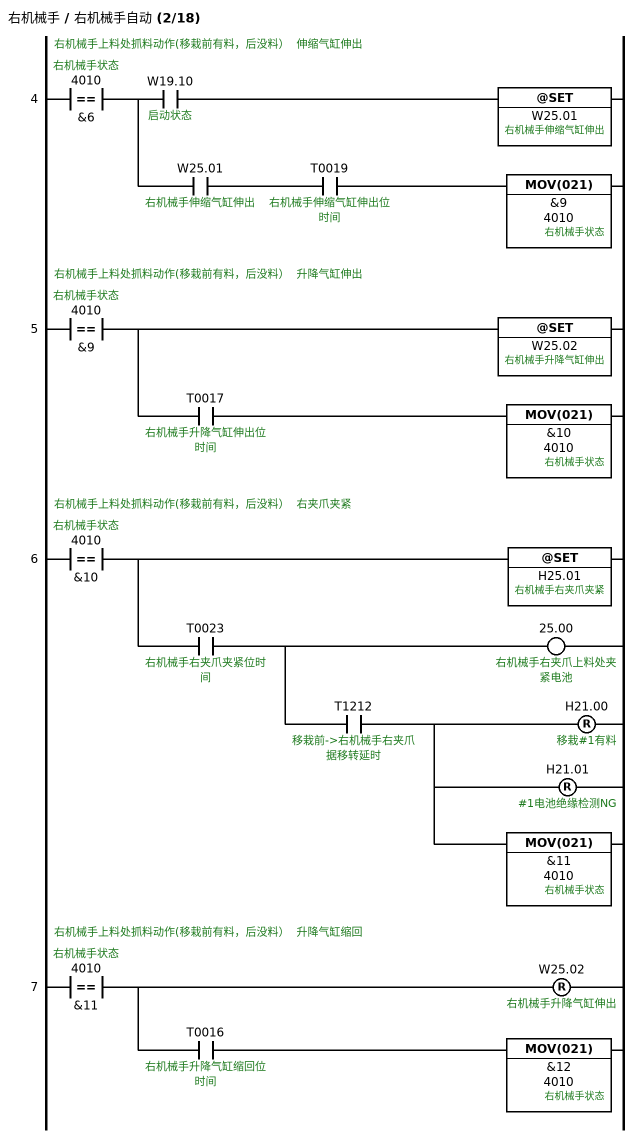
; rung 4: 右机械手上料处抓料动作(移栽前有料，后没料）  伸缩气缸伸出
LD=(300) 4010 &6  ; 右机械手状态
OUT TR0
AND W19.10  ; 启动状态
@SET W25.01  ; 右机械手伸缩气缸伸出
LD TR0
AND W25.01  ; 右机械手伸缩气缸伸出
AND T0019  ; 右机械手伸缩气缸伸出位时间
MOV(021) &9 4010  ; 右机械手状态
; rung 5: 右机械手上料处抓料动作(移栽前有料，后没料）  升降气缸伸出
LD=(300) 4010 &9  ; 右机械手状态
@SET W25.02  ; 右机械手升降气缸伸出
AND T0017  ; 右机械手升降气缸伸出位时间
MOV(021) &10 4010  ; 右机械手状态
; rung 6: 右机械手上料处抓料动作(移栽前有料，后没料）  右夹爪夹紧
LD=(300) 4010 &10  ; 右机械手状态
@SET H25.01  ; 右机械手右夹爪夹紧
AND T0023  ; 右机械手右夹爪夹紧位时间
OUT 25.00  ; 右机械手右夹爪上料处夹紧电池
AND T1212  ; 移栽前->右机械手右夹爪据移转延时
RSET H21.00  ; 移栽#1有料
RSET H21.01  ; #1电池绝缘检测NG
MOV(021) &11 4010  ; 右机械手状态
; rung 7: 右机械手上料处抓料动作(移栽前有料，后没料）  升降气缸缩回
LD=(300) 4010 &11  ; 右机械手状态
RSET W25.02  ; 右机械手升降气缸伸出
AND T0016  ; 右机械手升降气缸缩回位时间
MOV(021) &12 4010  ; 右机械手状态

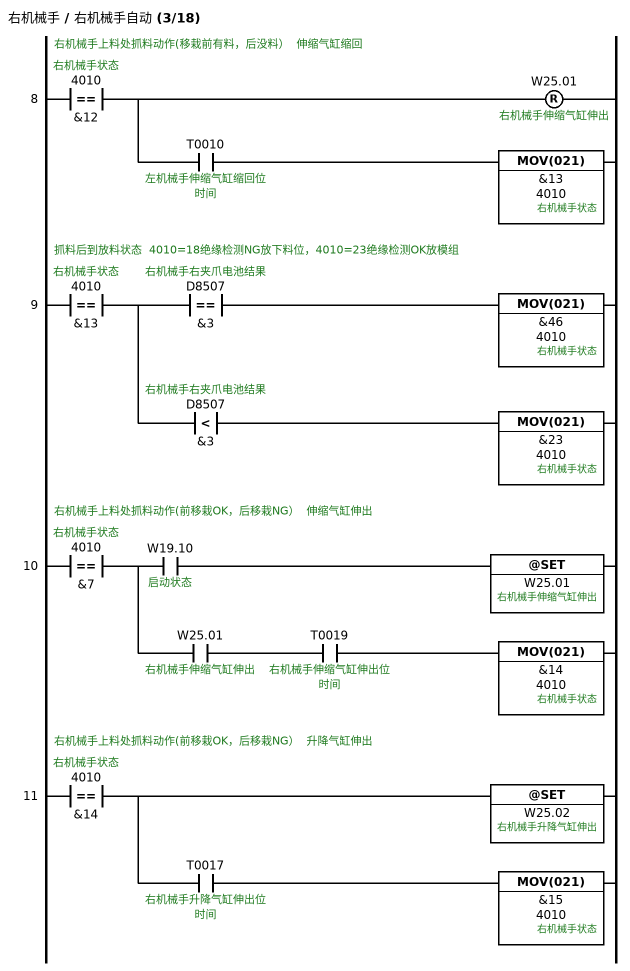
; rung 8: 右机械手上料处抓料动作(移栽前有料，后没料）  伸缩气缸缩回
LD=(300) 4010 &12  ; 右机械手状态
RSET W25.01  ; 右机械手伸缩气缸伸出
AND T0010  ; 左机械手伸缩气缸缩回位时间
MOV(021) &13 4010  ; 右机械手状态
; rung 9: 抓料后到放料状态  4010=18绝缘检测NG放下料位，4010=23绝缘检测OK放模组
LD=(300) 4010 &13  ; 右机械手状态
OUT TR0
AND=(300) D8507 &3  ; 右机械手右夹爪电池结果
MOV(021) &46 4010  ; 右机械手状态
LD TR0
AND<(310) D8507 &3  ; 右机械手右夹爪电池结果
MOV(021) &23 4010  ; 右机械手状态
; rung 10: 右机械手上料处抓料动作(前移栽OK，后移栽NG）  伸缩气缸伸出
LD=(300) 4010 &7  ; 右机械手状态
OUT TR0
AND W19.10  ; 启动状态
@SET W25.01  ; 右机械手伸缩气缸伸出
LD TR0
AND W25.01  ; 右机械手伸缩气缸伸出
AND T0019  ; 右机械手伸缩气缸伸出位时间
MOV(021) &14 4010  ; 右机械手状态
; rung 11: 右机械手上料处抓料动作(前移栽OK，后移栽NG）  升降气缸伸出
LD=(300) 4010 &14  ; 右机械手状态
@SET W25.02  ; 右机械手升降气缸伸出
AND T0017  ; 右机械手升降气缸伸出位时间
MOV(021) &15 4010  ; 右机械手状态

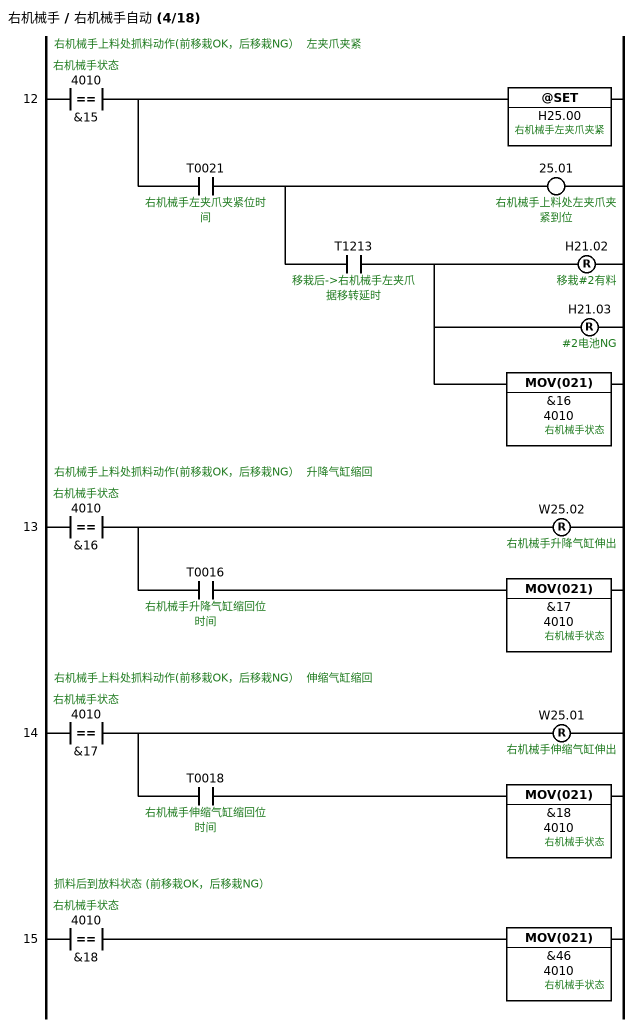
; rung 12: 右机械手上料处抓料动作(前移栽OK，后移栽NG）  左夹爪夹紧
LD=(300) 4010 &15  ; 右机械手状态
@SET H25.00  ; 右机械手左夹爪夹紧
AND T0021  ; 右机械手左夹爪夹紧位时间
OUT 25.01  ; 右机械手上料处左夹爪夹紧到位
AND T1213  ; 移栽后->右机械手左夹爪据移转延时
RSET H21.02  ; 移栽#2有料
RSET H21.03  ; #2电池NG
MOV(021) &16 4010  ; 右机械手状态
; rung 13: 右机械手上料处抓料动作(前移栽OK，后移栽NG）  升降气缸缩回
LD=(300) 4010 &16  ; 右机械手状态
RSET W25.02  ; 右机械手升降气缸伸出
AND T0016  ; 右机械手升降气缸缩回位时间
MOV(021) &17 4010  ; 右机械手状态
; rung 14: 右机械手上料处抓料动作(前移栽OK，后移栽NG）  伸缩气缸缩回
LD=(300) 4010 &17  ; 右机械手状态
RSET W25.01  ; 右机械手伸缩气缸伸出
AND T0018  ; 右机械手伸缩气缸缩回位时间
MOV(021) &18 4010  ; 右机械手状态
; rung 15: 抓料后到放料状态 (前移栽OK，后移栽NG）
LD=(300) 4010 &18  ; 右机械手状态
MOV(021) &46 4010  ; 右机械手状态

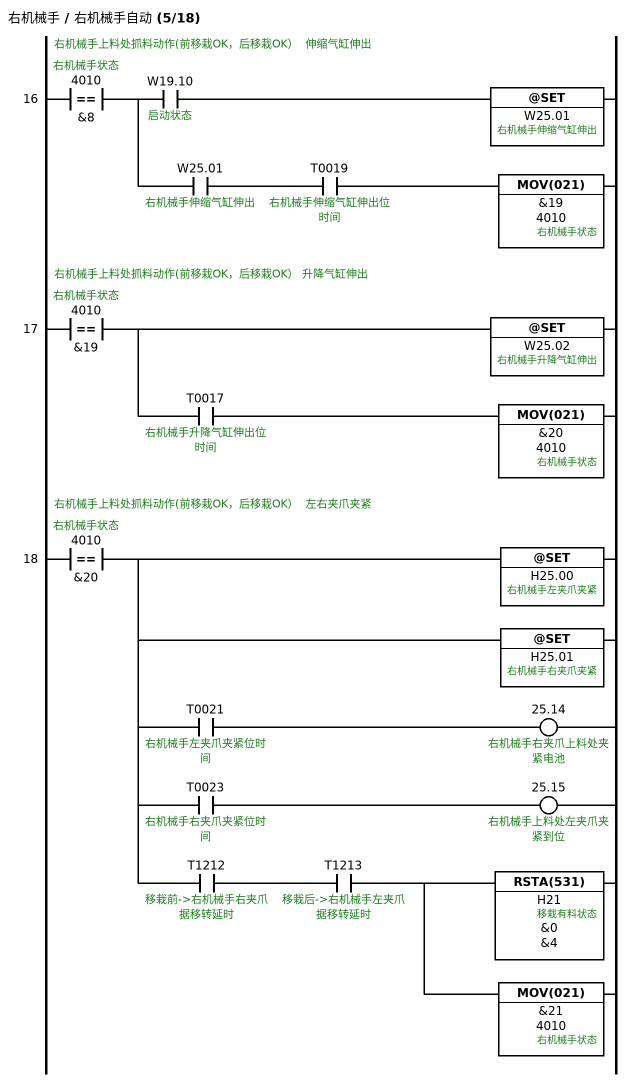
; rung 16: 右机械手上料处抓料动作(前移栽OK，后移栽OK）  伸缩气缸伸出
LD=(300) 4010 &8  ; 右机械手状态
OUT TR0
AND W19.10  ; 启动状态
@SET W25.01  ; 右机械手伸缩气缸伸出
LD TR0
AND W25.01  ; 右机械手伸缩气缸伸出
AND T0019  ; 右机械手伸缩气缸伸出位时间
MOV(021) &19 4010  ; 右机械手状态
; rung 17: 右机械手上料处抓料动作(前移栽OK，后移栽OK） 升降气缸伸出
LD=(300) 4010 &19  ; 右机械手状态
@SET W25.02  ; 右机械手升降气缸伸出
AND T0017  ; 右机械手升降气缸伸出位时间
MOV(021) &20 4010  ; 右机械手状态
; rung 18: 右机械手上料处抓料动作(前移栽OK，后移栽OK）  左右夹爪夹紧
LD=(300) 4010 &20  ; 右机械手状态
OUT TR0
@SET H25.00  ; 右机械手左夹爪夹紧
@SET H25.01  ; 右机械手右夹爪夹紧
AND T0021  ; 右机械手左夹爪夹紧位时间
OUT 25.14  ; 右机械手右夹爪上料处夹紧电池
LD TR0
AND T0023  ; 右机械手右夹爪夹紧位时间
OUT 25.15  ; 右机械手上料处左夹爪夹紧到位
LD TR0
AND T1212  ; 移栽前->右机械手右夹爪据移转延时
AND T1213  ; 移栽后->右机械手左夹爪据移转延时
RSTA(531) H21 &0 &4  ; 移栽有料状态
MOV(021) &21 4010  ; 右机械手状态

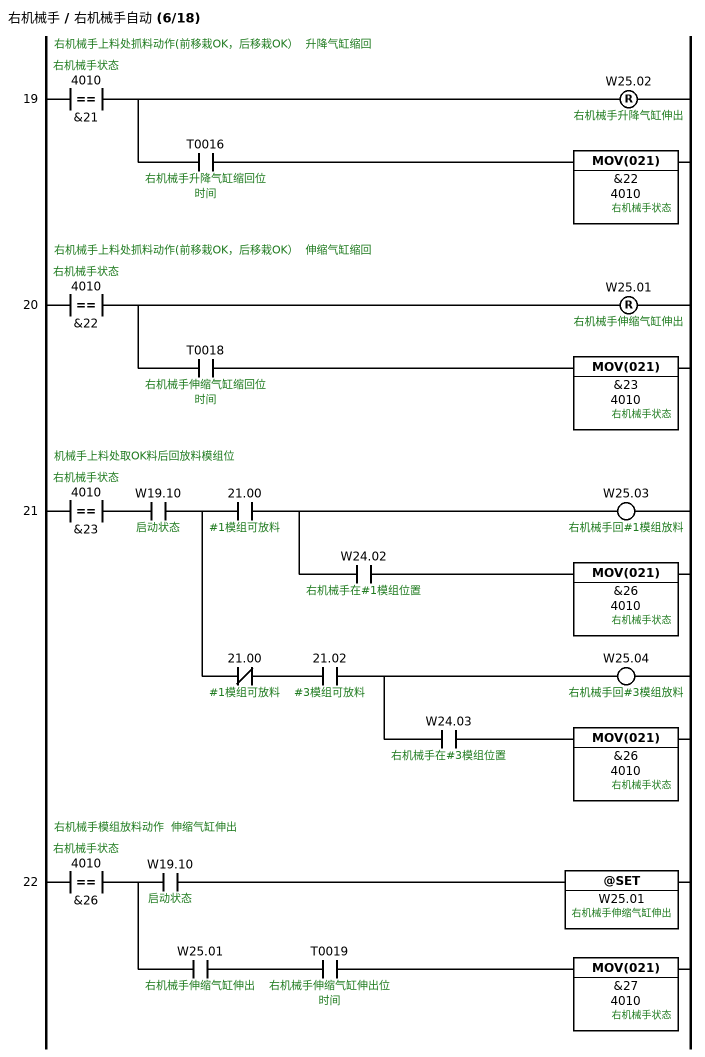
; rung 19: 右机械手上料处抓料动作(前移栽OK，后移栽OK）  升降气缸缩回
LD=(300) 4010 &21  ; 右机械手状态
RSET W25.02  ; 右机械手升降气缸伸出
AND T0016  ; 右机械手升降气缸缩回位时间
MOV(021) &22 4010  ; 右机械手状态
; rung 20: 右机械手上料处抓料动作(前移栽OK，后移栽OK）  伸缩气缸缩回
LD=(300) 4010 &22  ; 右机械手状态
RSET W25.01  ; 右机械手伸缩气缸伸出
AND T0018  ; 右机械手伸缩气缸缩回位时间
MOV(021) &23 4010  ; 右机械手状态
; rung 21: 机械手上料处取OK料后回放料模组位
LD=(300) 4010 &23  ; 右机械手状态
AND W19.10  ; 启动状态
OUT TR0
AND 21.00  ; #1模组可放料
OUT W25.03  ; 右机械手回#1模组放料
AND W24.02  ; 右机械手在#1模组位置
MOV(021) &26 4010  ; 右机械手状态
LD TR0
ANDNOT 21.00  ; #1模组可放料
AND 21.02  ; #3模组可放料
OUT W25.04  ; 右机械手回#3模组放料
AND W24.03  ; 右机械手在#3模组位置
MOV(021) &26 4010  ; 右机械手状态
; rung 22: 右机械手模组放料动作  伸缩气缸伸出
LD=(300) 4010 &26  ; 右机械手状态
OUT TR0
AND W19.10  ; 启动状态
@SET W25.01  ; 右机械手伸缩气缸伸出
LD TR0
AND W25.01  ; 右机械手伸缩气缸伸出
AND T0019  ; 右机械手伸缩气缸伸出位时间
MOV(021) &27 4010  ; 右机械手状态

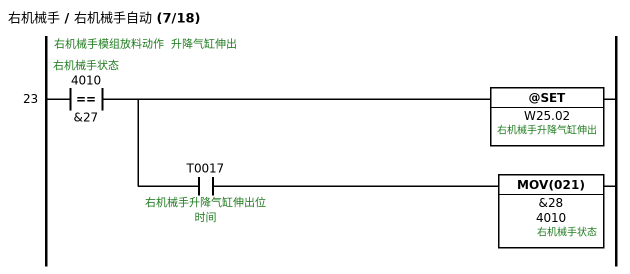
; rung 23: 右机械手模组放料动作  升降气缸伸出
LD=(300) 4010 &27  ; 右机械手状态
@SET W25.02  ; 右机械手升降气缸伸出
AND T0017  ; 右机械手升降气缸伸出位时间
MOV(021) &28 4010  ; 右机械手状态

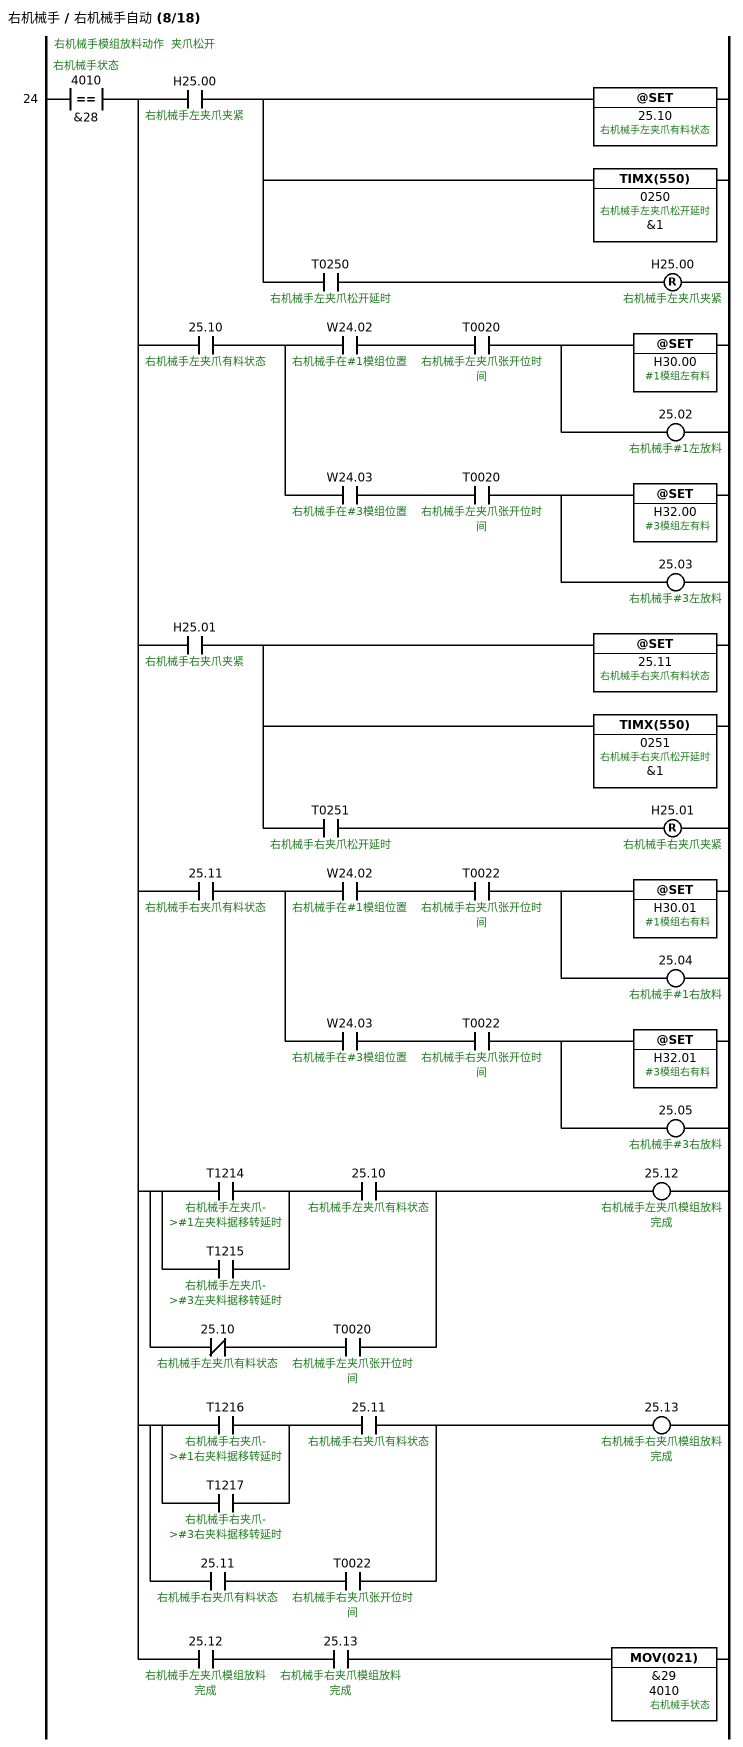
; rung 24: 右机械手模组放料动作  夹爪松开
LD=(300) 4010 &28  ; 右机械手状态
OUT TR0
AND H25.00  ; 右机械手左夹爪夹紧
@SET 25.10  ; 右机械手左夹爪有料状态
TIMX(550) 0250 &1  ; 右机械手左夹爪松开延时
AND T0250  ; 右机械手左夹爪松开延时
RSET H25.00  ; 右机械手左夹爪夹紧
LD TR0
AND 25.10  ; 右机械手左夹爪有料状态
OUT TR1
AND W24.02  ; 右机械手在#1模组位置
AND T0020  ; 右机械手左夹爪张开位时间
@SET H30.00  ; #1模组左有料
OUT 25.02  ; 右机械手#1左放料
LD TR1
AND W24.03  ; 右机械手在#3模组位置
AND T0020  ; 右机械手左夹爪张开位时间
@SET H32.00  ; #3模组左有料
OUT 25.03  ; 右机械手#3左放料
LD TR0
AND H25.01  ; 右机械手右夹爪夹紧
@SET 25.11  ; 右机械手右夹爪有料状态
TIMX(550) 0251 &1  ; 右机械手右夹爪松开延时
AND T0251  ; 右机械手右夹爪松开延时
RSET H25.01  ; 右机械手右夹爪夹紧
LD TR0
AND 25.11  ; 右机械手右夹爪有料状态
OUT TR1
AND W24.02  ; 右机械手在#1模组位置
AND T0022  ; 右机械手右夹爪张开位时间
@SET H30.01  ; #1模组右有料
OUT 25.04  ; 右机械手#1右放料
LD TR1
AND W24.03  ; 右机械手在#3模组位置
AND T0022  ; 右机械手右夹爪张开位时间
@SET H32.01  ; #3模组右有料
OUT 25.05  ; 右机械手#3右放料
LD TR0
LD T1214  ; 右机械手左夹爪->#1左夹料据移转延时
OR T1215  ; 右机械手左夹爪->#3左夹料据移转延时
AND 25.10  ; 右机械手左夹爪有料状态
LDNOT 25.10  ; 右机械手左夹爪有料状态
AND T0020  ; 右机械手左夹爪张开位时间
ORLD
ANDLD
OUT 25.12  ; 右机械手左夹爪模组放料完成
LD TR0
LD T1216  ; 右机械手右夹爪->#1右夹料据移转延时
OR T1217  ; 右机械手右夹爪->#3右夹料据移转延时
AND 25.11  ; 右机械手右夹爪有料状态
LD 25.11  ; 右机械手右夹爪有料状态
AND T0022  ; 右机械手右夹爪张开位时间
ORLD
ANDLD
OUT 25.13  ; 右机械手右夹爪模组放料完成
LD TR0
AND 25.12  ; 右机械手左夹爪模组放料完成
AND 25.13  ; 右机械手右夹爪模组放料完成
MOV(021) &29 4010  ; 右机械手状态

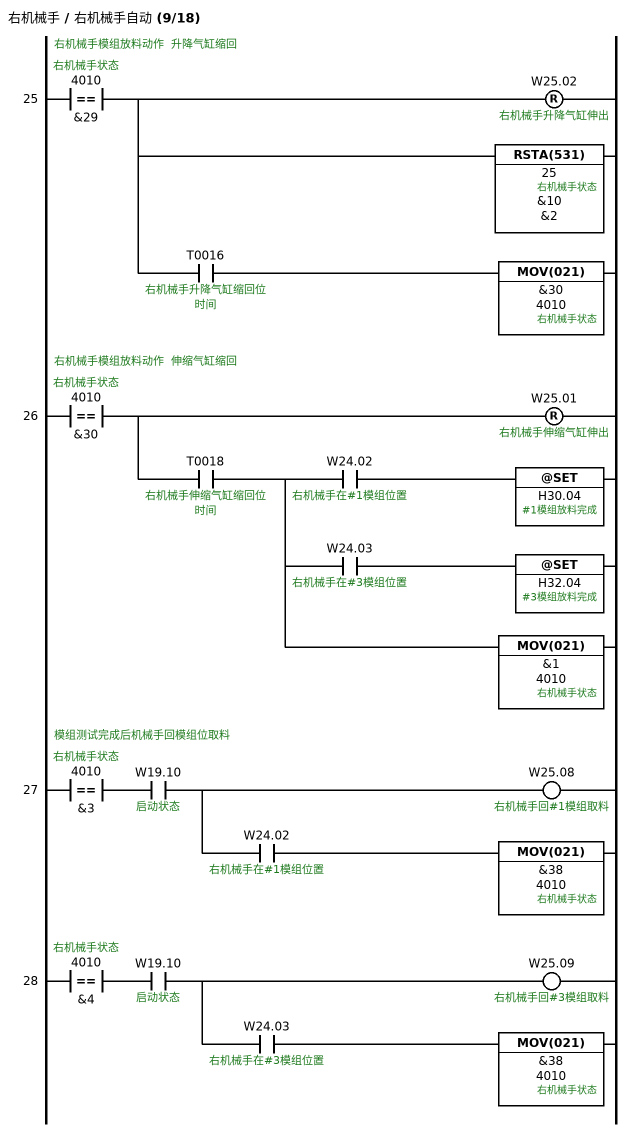
; rung 25: 右机械手模组放料动作  升降气缸缩回
LD=(300) 4010 &29  ; 右机械手状态
RSET W25.02  ; 右机械手升降气缸伸出
RSTA(531) 25 &10 &2  ; 右机械手状态
AND T0016  ; 右机械手升降气缸缩回位时间
MOV(021) &30 4010  ; 右机械手状态
; rung 26: 右机械手模组放料动作  伸缩气缸缩回
LD=(300) 4010 &30  ; 右机械手状态
RSET W25.01  ; 右机械手伸缩气缸伸出
AND T0018  ; 右机械手伸缩气缸缩回位时间
OUT TR0
AND W24.02  ; 右机械手在#1模组位置
@SET H30.04  ; #1模组放料完成
LD TR0
AND W24.03  ; 右机械手在#3模组位置
@SET H32.04  ; #3模组放料完成
LD TR0
MOV(021) &1 4010  ; 右机械手状态
; rung 27: 模组测试完成后机械手回模组位取料
LD=(300) 4010 &3  ; 右机械手状态
AND W19.10  ; 启动状态
OUT W25.08  ; 右机械手回#1模组取料
AND W24.02  ; 右机械手在#1模组位置
MOV(021) &38 4010  ; 右机械手状态
; rung 28
LD=(300) 4010 &4  ; 右机械手状态
AND W19.10  ; 启动状态
OUT W25.09  ; 右机械手回#3模组取料
AND W24.03  ; 右机械手在#3模组位置
MOV(021) &38 4010  ; 右机械手状态

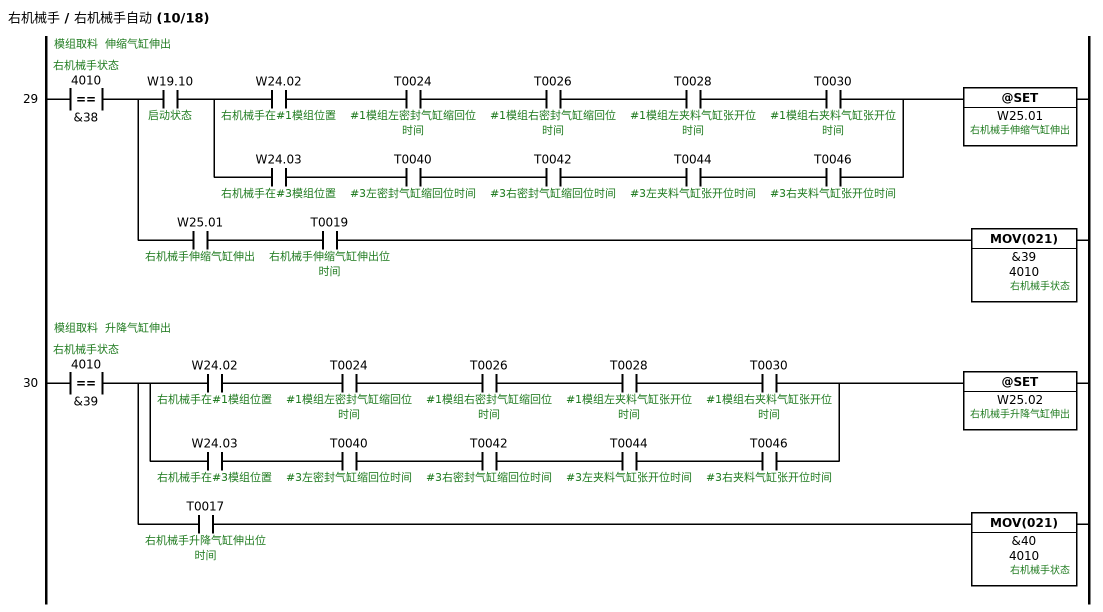
; rung 29: 模组取料  伸缩气缸伸出
LD=(300) 4010 &38  ; 右机械手状态
OUT TR0
AND W19.10  ; 启动状态
LD W24.02  ; 右机械手在#1模组位置
AND T0024  ; #1模组左密封气缸缩回位时间
AND T0026  ; #1模组右密封气缸缩回位时间
AND T0028  ; #1模组左夹料气缸张开位时间
AND T0030  ; #1模组右夹料气缸张开位时间
LD W24.03  ; 右机械手在#3模组位置
AND T0040  ; #3左密封气缸缩回位时间
AND T0042  ; #3右密封气缸缩回位时间
AND T0044  ; #3左夹料气缸张开位时间
AND T0046  ; #3右夹料气缸张开位时间
ORLD
ANDLD
@SET W25.01  ; 右机械手伸缩气缸伸出
LD TR0
AND W25.01  ; 右机械手伸缩气缸伸出
AND T0019  ; 右机械手伸缩气缸伸出位时间
MOV(021) &39 4010  ; 右机械手状态
; rung 30: 模组取料  升降气缸伸出
LD=(300) 4010 &39  ; 右机械手状态
OUT TR0
LD W24.02  ; 右机械手在#1模组位置
AND T0024  ; #1模组左密封气缸缩回位时间
AND T0026  ; #1模组右密封气缸缩回位时间
AND T0028  ; #1模组左夹料气缸张开位时间
AND T0030  ; #1模组右夹料气缸张开位时间
LD W24.03  ; 右机械手在#3模组位置
AND T0040  ; #3左密封气缸缩回位时间
AND T0042  ; #3右密封气缸缩回位时间
AND T0044  ; #3左夹料气缸张开位时间
AND T0046  ; #3右夹料气缸张开位时间
ORLD
ANDLD
@SET W25.02  ; 右机械手升降气缸伸出
LD TR0
AND T0017  ; 右机械手升降气缸伸出位时间
MOV(021) &40 4010  ; 右机械手状态

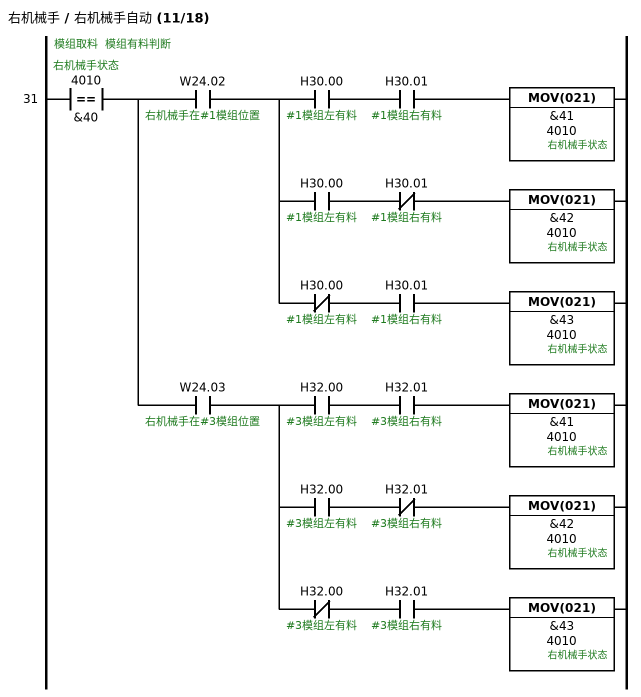
; rung 31: 模组取料  模组有料判断
LD=(300) 4010 &40  ; 右机械手状态
OUT TR0
AND W24.02  ; 右机械手在#1模组位置
OUT TR1
AND H30.00  ; #1模组左有料
AND H30.01  ; #1模组右有料
MOV(021) &41 4010  ; 右机械手状态
LD TR1
AND H30.00  ; #1模组左有料
ANDNOT H30.01  ; #1模组右有料
MOV(021) &42 4010  ; 右机械手状态
LD TR1
ANDNOT H30.00  ; #1模组左有料
AND H30.01  ; #1模组右有料
MOV(021) &43 4010  ; 右机械手状态
LD TR0
AND W24.03  ; 右机械手在#3模组位置
OUT TR0
AND H32.00  ; #3模组左有料
AND H32.01  ; #3模组右有料
MOV(021) &41 4010  ; 右机械手状态
LD TR0
AND H32.00  ; #3模组左有料
ANDNOT H32.01  ; #3模组右有料
MOV(021) &42 4010  ; 右机械手状态
LD TR0
ANDNOT H32.00  ; #3模组左有料
AND H32.01  ; #3模组右有料
MOV(021) &43 4010  ; 右机械手状态

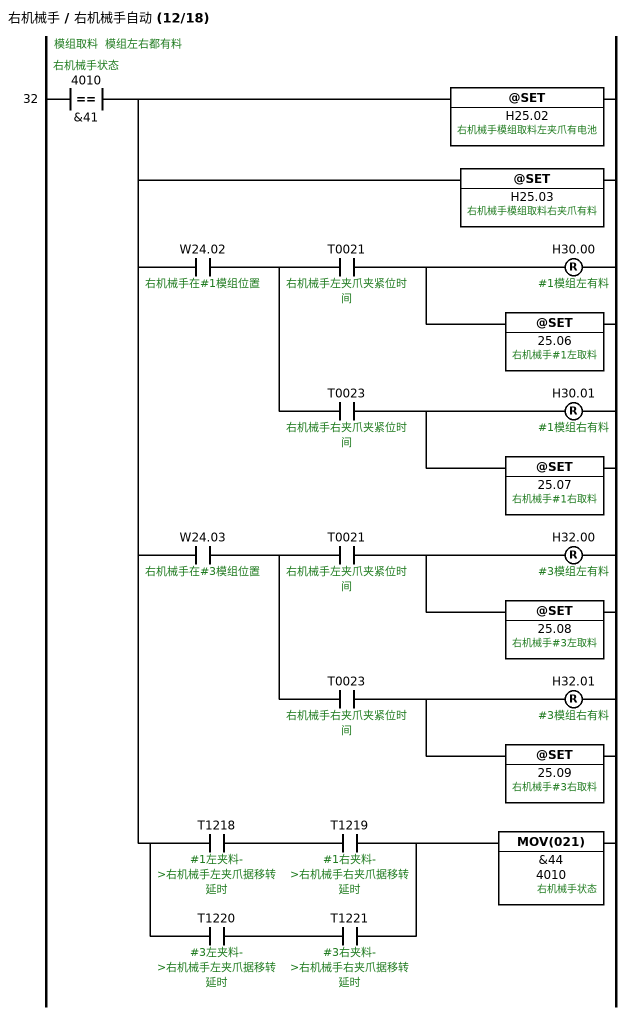
; rung 32: 模组取料  模组左右都有料
LD=(300) 4010 &41  ; 右机械手状态
OUT TR0
@SET H25.02  ; 右机械手模组取料左夹爪有电池
@SET H25.03  ; 右机械手模组取料右夹爪有料
AND W24.02  ; 右机械手在#1模组位置
OUT TR1
AND T0021  ; 右机械手左夹爪夹紧位时间
RSET H30.00  ; #1模组左有料
@SET 25.06  ; 右机械手#1左取料
LD TR1
AND T0023  ; 右机械手右夹爪夹紧位时间
RSET H30.01  ; #1模组右有料
@SET 25.07  ; 右机械手#1右取料
LD TR0
AND W24.03  ; 右机械手在#3模组位置
OUT TR1
AND T0021  ; 右机械手左夹爪夹紧位时间
RSET H32.00  ; #3模组左有料
@SET 25.08  ; 右机械手#3左取料
LD TR1
AND T0023  ; 右机械手右夹爪夹紧位时间
RSET H32.01  ; #3模组右有料
@SET 25.09  ; 右机械手#3右取料
LD TR0
LD T1218  ; #1左夹料->右机械手左夹爪据移转延时
AND T1219  ; #1右夹料->右机械手右夹爪据移转延时
LD T1220  ; #3左夹料->右机械手左夹爪据移转延时
AND T1221  ; #3右夹料->右机械手右夹爪据移转延时
ORLD
ANDLD
MOV(021) &44 4010  ; 右机械手状态

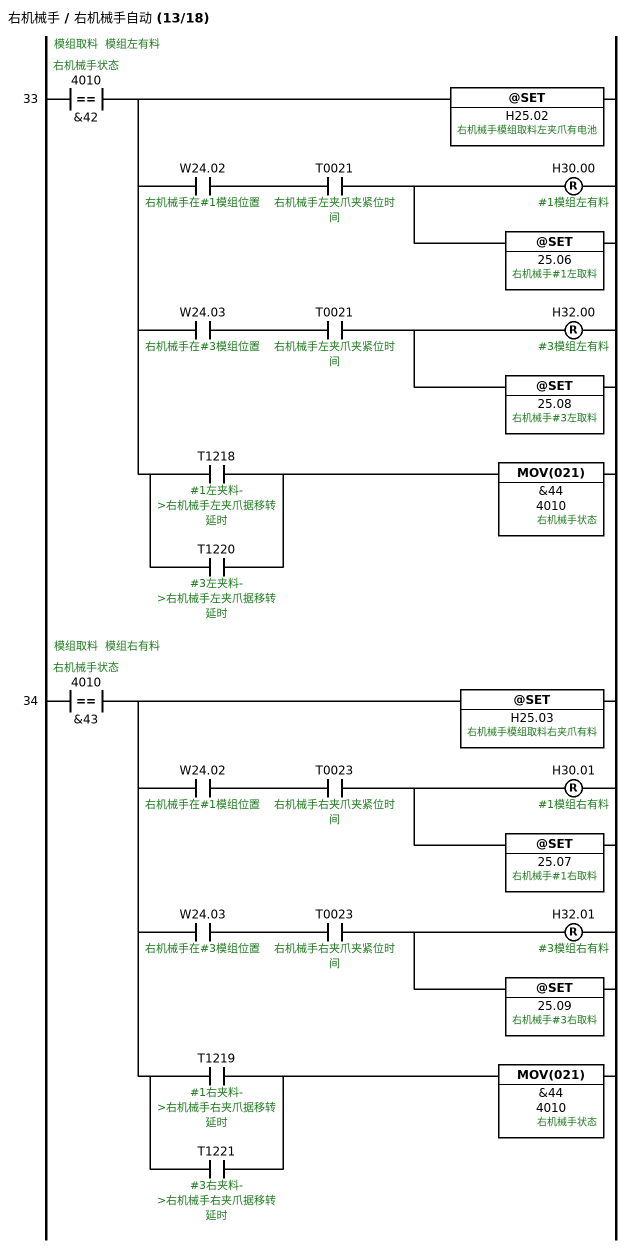
; rung 33: 模组取料  模组左有料
LD=(300) 4010 &42  ; 右机械手状态
OUT TR0
@SET H25.02  ; 右机械手模组取料左夹爪有电池
AND W24.02  ; 右机械手在#1模组位置
AND T0021  ; 右机械手左夹爪夹紧位时间
RSET H30.00  ; #1模组左有料
@SET 25.06  ; 右机械手#1左取料
LD TR0
AND W24.03  ; 右机械手在#3模组位置
AND T0021  ; 右机械手左夹爪夹紧位时间
RSET H32.00  ; #3模组左有料
@SET 25.08  ; 右机械手#3左取料
LD TR0
LD T1218  ; #1左夹料->右机械手左夹爪据移转延时
OR T1220  ; #3左夹料->右机械手左夹爪据移转延时
ANDLD
MOV(021) &44 4010  ; 右机械手状态
; rung 34: 模组取料  模组右有料
LD=(300) 4010 &43  ; 右机械手状态
OUT TR0
@SET H25.03  ; 右机械手模组取料右夹爪有料
AND W24.02  ; 右机械手在#1模组位置
AND T0023  ; 右机械手右夹爪夹紧位时间
RSET H30.01  ; #1模组右有料
@SET 25.07  ; 右机械手#1右取料
LD TR0
AND W24.03  ; 右机械手在#3模组位置
AND T0023  ; 右机械手右夹爪夹紧位时间
RSET H32.01  ; #3模组右有料
@SET 25.09  ; 右机械手#3右取料
LD TR0
LD T1219  ; #1右夹料->右机械手右夹爪据移转延时
OR T1221  ; #3右夹料->右机械手右夹爪据移转延时
ANDLD
MOV(021) &44 4010  ; 右机械手状态

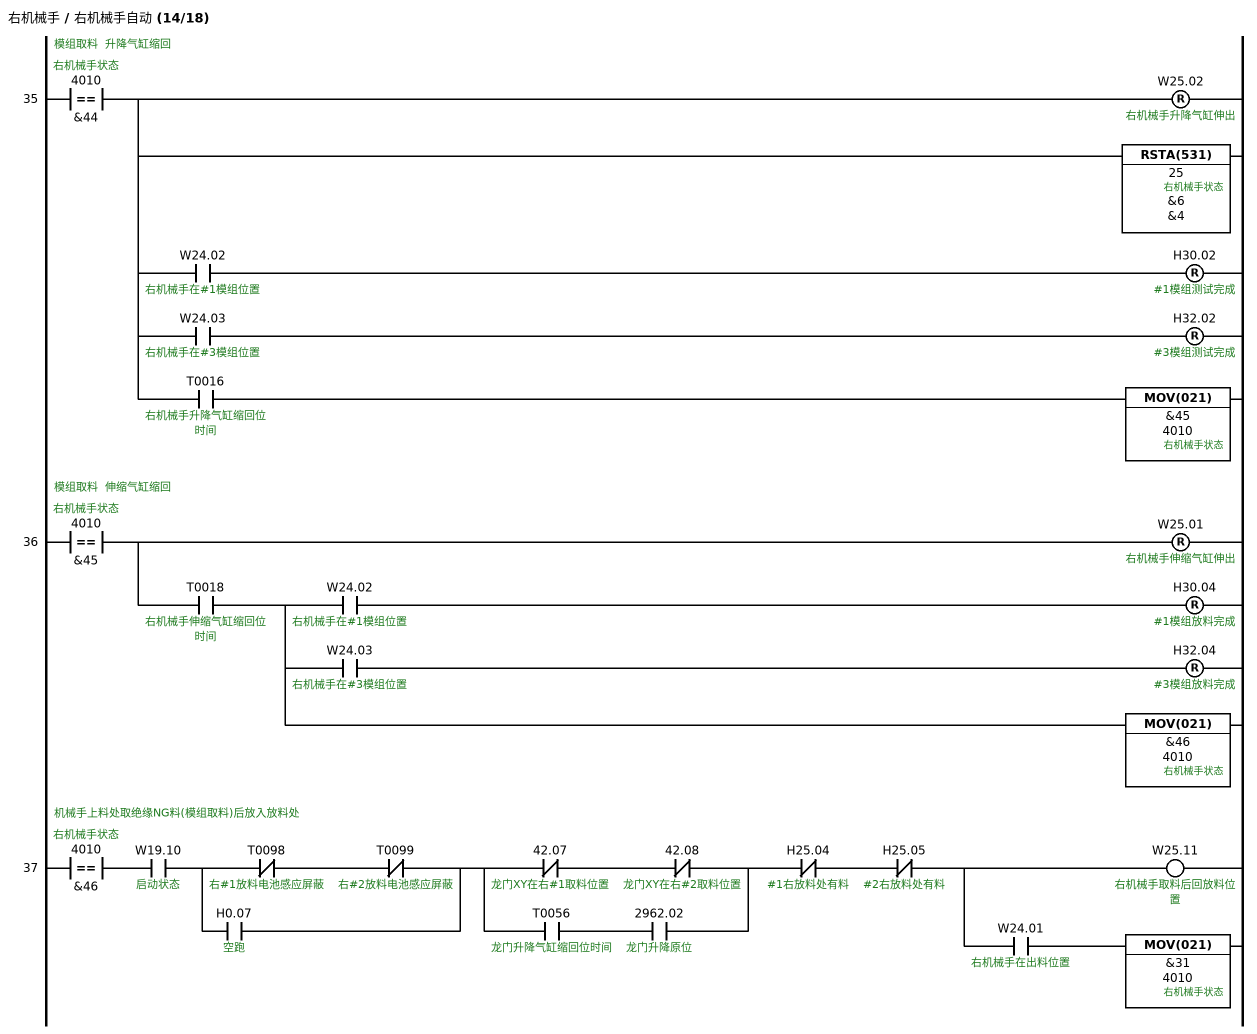
; rung 35: 模组取料  升降气缸缩回
LD=(300) 4010 &44  ; 右机械手状态
OUT TR0
RSET W25.02  ; 右机械手升降气缸伸出
RSTA(531) 25 &6 &4  ; 右机械手状态
AND W24.02  ; 右机械手在#1模组位置
RSET H30.02  ; #1模组测试完成
LD TR0
AND W24.03  ; 右机械手在#3模组位置
RSET H32.02  ; #3模组测试完成
LD TR0
AND T0016  ; 右机械手升降气缸缩回位时间
MOV(021) &45 4010  ; 右机械手状态
; rung 36: 模组取料  伸缩气缸缩回
LD=(300) 4010 &45  ; 右机械手状态
RSET W25.01  ; 右机械手伸缩气缸伸出
AND T0018  ; 右机械手伸缩气缸缩回位时间
OUT TR0
AND W24.02  ; 右机械手在#1模组位置
RSET H30.04  ; #1模组放料完成
LD TR0
AND W24.03  ; 右机械手在#3模组位置
RSET H32.04  ; #3模组放料完成
LD TR0
MOV(021) &46 4010  ; 右机械手状态
; rung 37: 机械手上料处取绝缘NG料(模组取料)后放入放料处
LD=(300) 4010 &46  ; 右机械手状态
AND W19.10  ; 启动状态
LDNOT T0098  ; 右#1放料电池感应屏蔽
ANDNOT T0099  ; 右#2放料电池感应屏蔽
OR H0.07  ; 空跑
ANDLD
LDNOT 42.07  ; 龙门XY在右#1取料位置
ANDNOT 42.08  ; 龙门XY在右#2取料位置
LD T0056  ; 龙门升降气缸缩回位时间
AND 2962.02  ; 龙门升降原位
ORLD
ANDLD
ANDNOT H25.04  ; #1右放料处有料
ANDNOT H25.05  ; #2右放料处有料
OUT W25.11  ; 右机械手取料后回放料位置
AND W24.01  ; 右机械手在出料位置
MOV(021) &31 4010  ; 右机械手状态

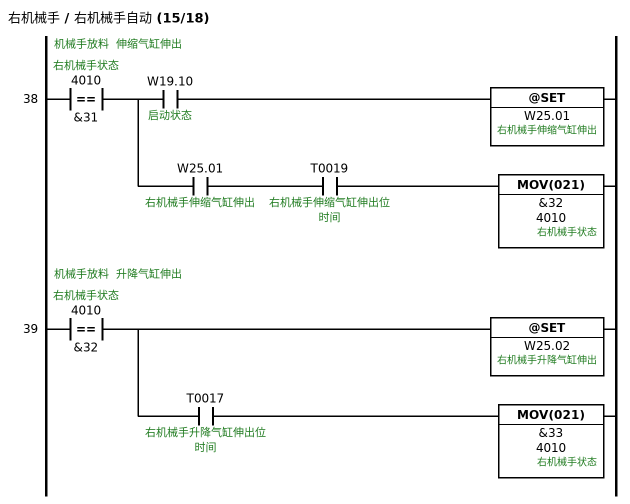
; rung 38: 机械手放料  伸缩气缸伸出
LD=(300) 4010 &31  ; 右机械手状态
OUT TR0
AND W19.10  ; 启动状态
@SET W25.01  ; 右机械手伸缩气缸伸出
LD TR0
AND W25.01  ; 右机械手伸缩气缸伸出
AND T0019  ; 右机械手伸缩气缸伸出位时间
MOV(021) &32 4010  ; 右机械手状态
; rung 39: 机械手放料  升降气缸伸出
LD=(300) 4010 &32  ; 右机械手状态
@SET W25.02  ; 右机械手升降气缸伸出
AND T0017  ; 右机械手升降气缸伸出位时间
MOV(021) &33 4010  ; 右机械手状态

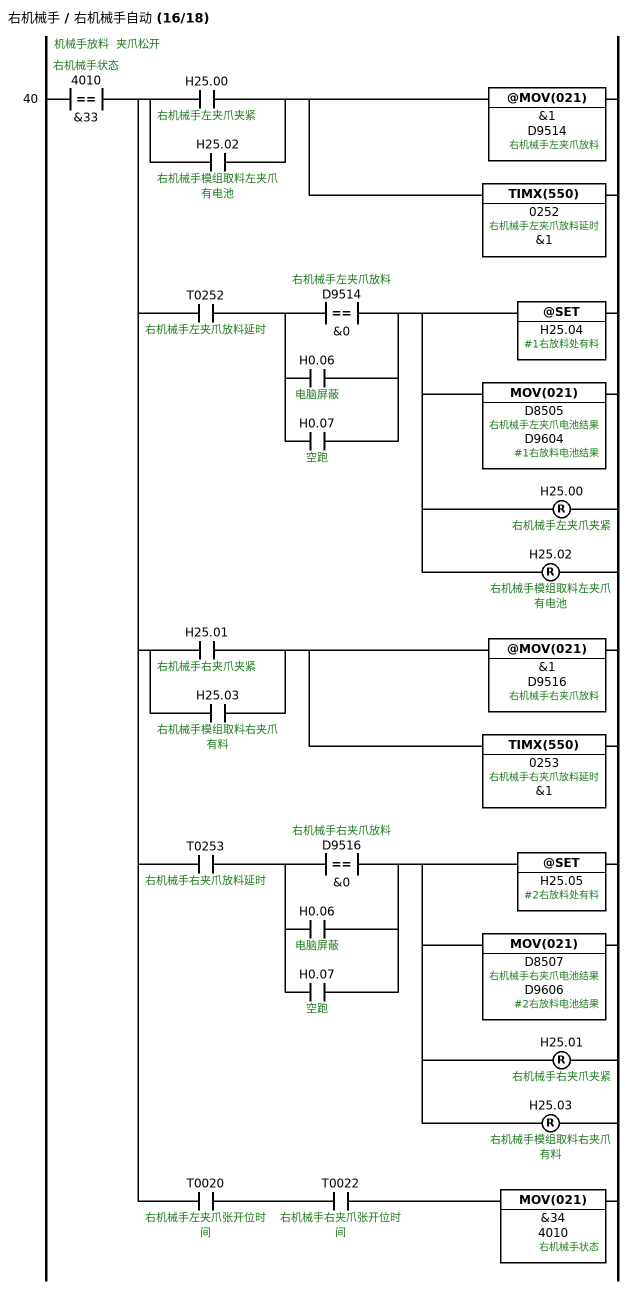
; rung 40: 机械手放料  夹爪松开
LD=(300) 4010 &33  ; 右机械手状态
OUT TR0
LD H25.00  ; 右机械手左夹爪夹紧
OR H25.02  ; 右机械手模组取料左夹爪有电池
ANDLD
@MOV(021) &1 D9514  ; 右机械手左夹爪放料
TIMX(550) 0252 &1  ; 右机械手左夹爪放料延时
LD TR0
AND T0252  ; 右机械手左夹爪放料延时
LD=(300) D9514 &0  ; 右机械手左夹爪放料
OR H0.06  ; 电脑屏蔽
OR H0.07  ; 空跑
ANDLD
@SET H25.04  ; #1右放料处有料
MOV(021) D8505 D9604  ; 右机械手左夹爪电池结果, #1右放料电池结果
RSET H25.00  ; 右机械手左夹爪夹紧
RSET H25.02  ; 右机械手模组取料左夹爪有电池
LD TR0
LD H25.01  ; 右机械手右夹爪夹紧
OR H25.03  ; 右机械手模组取料右夹爪有料
ANDLD
@MOV(021) &1 D9516  ; 右机械手右夹爪放料
TIMX(550) 0253 &1  ; 右机械手右夹爪放料延时
LD TR0
AND T0253  ; 右机械手右夹爪放料延时
LD=(300) D9516 &0  ; 右机械手右夹爪放料
OR H0.06  ; 电脑屏蔽
OR H0.07  ; 空跑
ANDLD
@SET H25.05  ; #2右放料处有料
MOV(021) D8507 D9606  ; 右机械手右夹爪电池结果, #2右放料电池结果
RSET H25.01  ; 右机械手右夹爪夹紧
RSET H25.03  ; 右机械手模组取料右夹爪有料
LD TR0
AND T0020  ; 右机械手左夹爪张开位时间
AND T0022  ; 右机械手右夹爪张开位时间
MOV(021) &34 4010  ; 右机械手状态

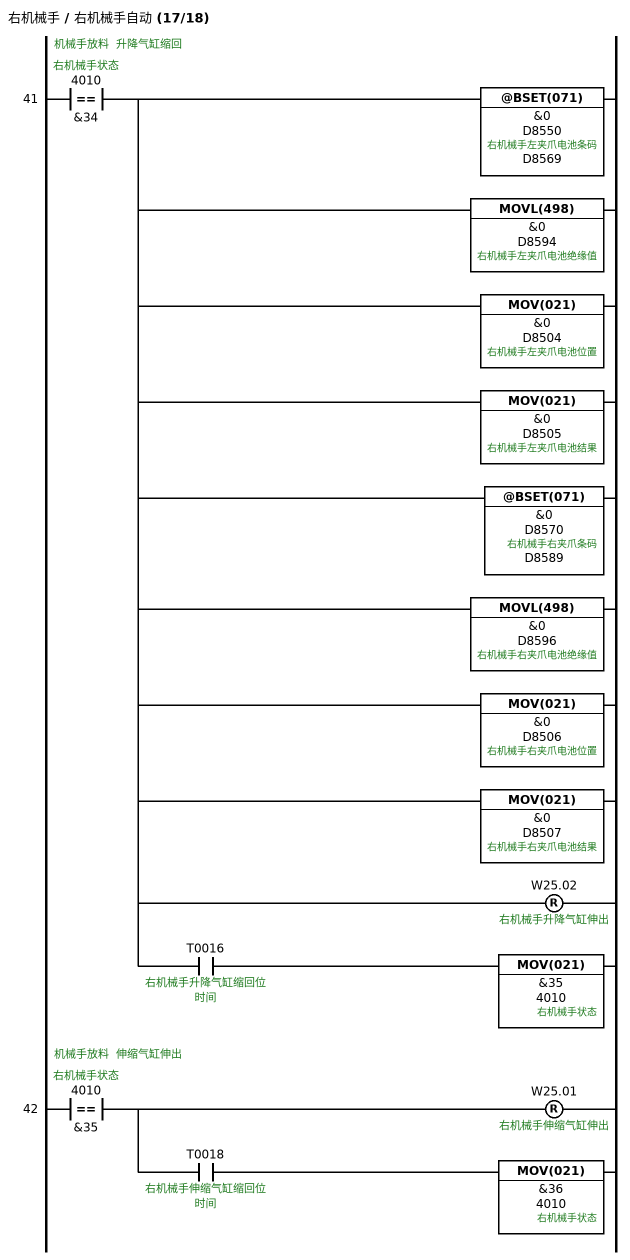
; rung 41: 机械手放料  升降气缸缩回
LD=(300) 4010 &34  ; 右机械手状态
@BSET(071) &0 D8550 D8569  ; 右机械手左夹爪电池条码
MOVL(498) &0 D8594  ; 右机械手左夹爪电池绝缘值
MOV(021) &0 D8504  ; 右机械手左夹爪电池位置
MOV(021) &0 D8505  ; 右机械手左夹爪电池结果
@BSET(071) &0 D8570 D8589  ; 右机械手右夹爪条码
MOVL(498) &0 D8596  ; 右机械手右夹爪电池绝缘值
MOV(021) &0 D8506  ; 右机械手右夹爪电池位置
MOV(021) &0 D8507  ; 右机械手右夹爪电池结果
RSET W25.02  ; 右机械手升降气缸伸出
AND T0016  ; 右机械手升降气缸缩回位时间
MOV(021) &35 4010  ; 右机械手状态
; rung 42: 机械手放料  伸缩气缸伸出
LD=(300) 4010 &35  ; 右机械手状态
RSET W25.01  ; 右机械手伸缩气缸伸出
AND T0018  ; 右机械手伸缩气缸缩回位时间
MOV(021) &36 4010  ; 右机械手状态

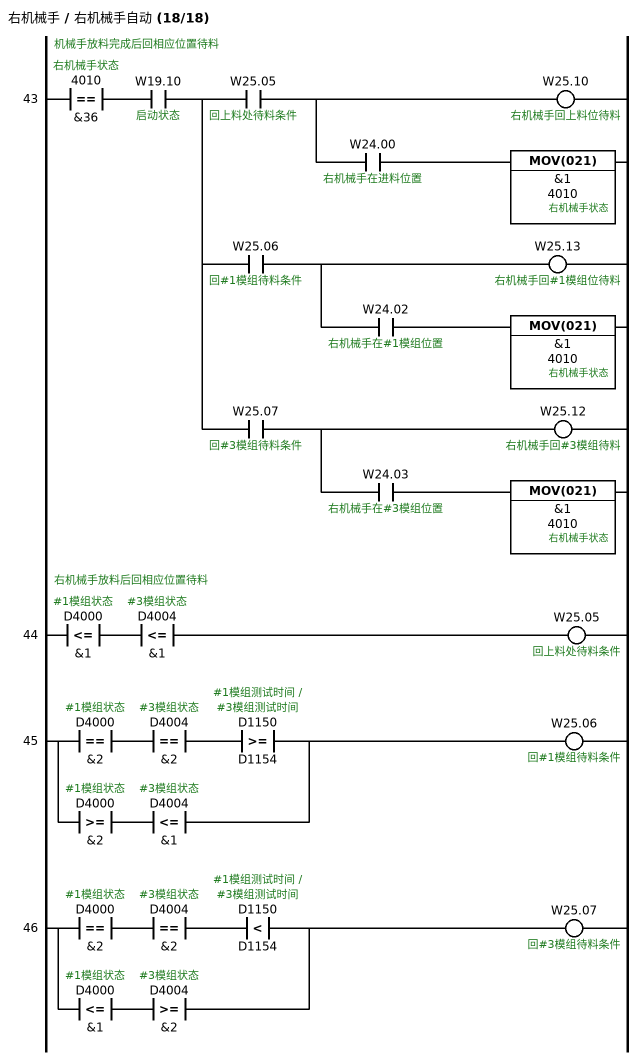
; rung 43: 机械手放料完成后回相应位置待料
LD=(300) 4010 &36  ; 右机械手状态
AND W19.10  ; 启动状态
OUT TR0
AND W25.05  ; 回上料处待料条件
OUT W25.10  ; 右机械手回上料位待料
AND W24.00  ; 右机械手在进料位置
MOV(021) &1 4010  ; 右机械手状态
LD TR0
AND W25.06  ; 回#1模组待料条件
OUT W25.13  ; 右机械手回#1模组位待料
AND W24.02  ; 右机械手在#1模组位置
MOV(021) &1 4010  ; 右机械手状态
LD TR0
AND W25.07  ; 回#3模组待料条件
OUT W25.12  ; 右机械手回#3模组待料
AND W24.03  ; 右机械手在#3模组位置
MOV(021) &1 4010  ; 右机械手状态
; rung 44: 右机械手放料后回相应位置待料
LD<=(315) D4000 &1  ; #1模组状态
AND<=(315) D4004 &1  ; #3模组状态
OUT W25.05  ; 回上料处待料条件
; rung 45
LD=(300) D4000 &2  ; #1模组状态
AND=(300) D4004 &2  ; #3模组状态
AND>=(325) D1150 D1154  ; #1模组测试时间, #3模组测试时间
LD>=(325) D4000 &2  ; #1模组状态
AND<=(315) D4004 &1  ; #3模组状态
ORLD
OUT W25.06  ; 回#1模组待料条件
; rung 46
LD=(300) D4000 &2  ; #1模组状态
AND=(300) D4004 &2  ; #3模组状态
AND<(310) D1150 D1154  ; #1模组测试时间, #3模组测试时间
LD<=(315) D4000 &1  ; #1模组状态
AND>=(325) D4004 &2  ; #3模组状态
ORLD
OUT W25.07  ; 回#3模组待料条件

### Section 伺服参数

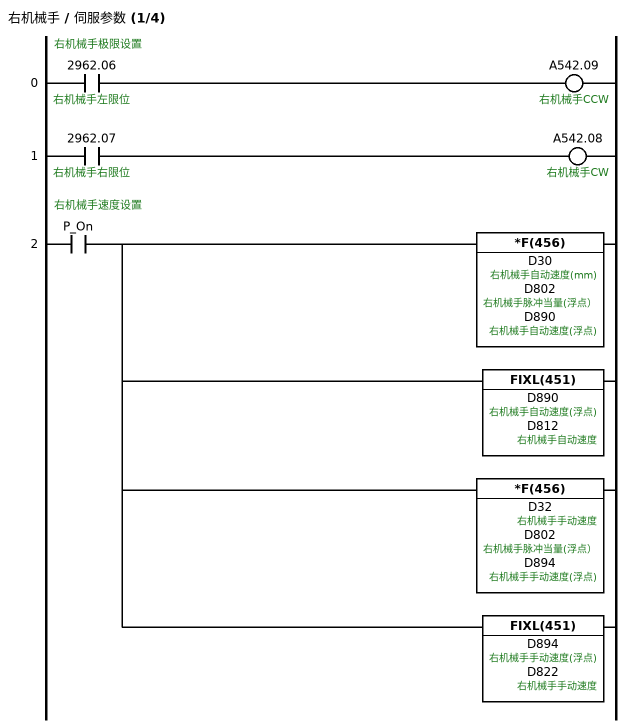
; rung 0: 右机械手极限设置
LD 2962.06  ; 右机械手左限位
OUT A542.09  ; 右机械手CCW
; rung 1
LD 2962.07  ; 右机械手右限位
OUT A542.08  ; 右机械手CW
; rung 2: 右机械手速度设置
LD P_On
*F(456) D30 D802 D890  ; 右机械手自动速度(mm), 右机械手脉冲当量(浮点）, 右机械手自动速度(浮点)
FIXL(451) D890 D812  ; 右机械手自动速度(浮点), 右机械手自动速度
*F(456) D32 D802 D894  ; 右机械手手动速度, 右机械手脉冲当量(浮点）, 右机械手手动速度(浮点)
FIXL(451) D894 D822  ; 右机械手手动速度(浮点), 右机械手手动速度

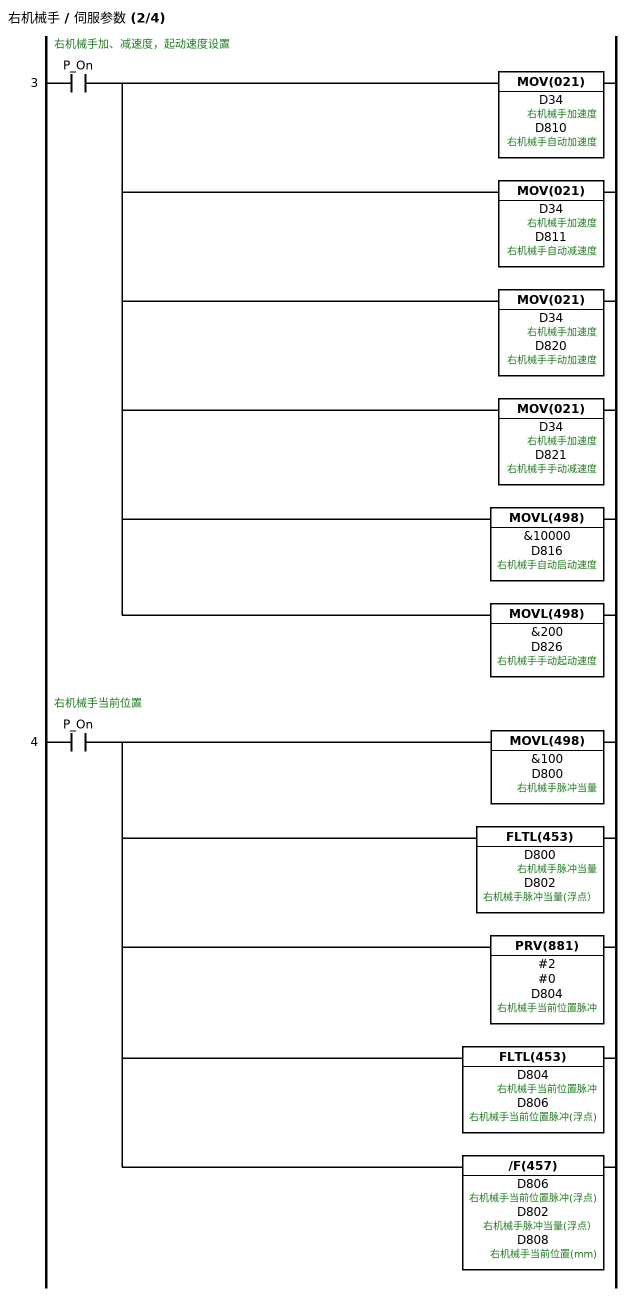
; rung 3: 右机械手加、减速度，起动速度设置
LD P_On
MOV(021) D34 D810  ; 右机械手加速度, 右机械手自动加速度
MOV(021) D34 D811  ; 右机械手加速度, 右机械手自动减速度
MOV(021) D34 D820  ; 右机械手加速度, 右机械手手动加速度
MOV(021) D34 D821  ; 右机械手加速度, 右机械手手动减速度
MOVL(498) &10000 D816  ; 右机械手自动启动速度
MOVL(498) &200 D826  ; 右机械手手动起动速度
; rung 4: 右机械手当前位置
LD P_On
MOVL(498) &100 D800  ; 右机械手脉冲当量
FLTL(453) D800 D802  ; 右机械手脉冲当量, 右机械手脉冲当量(浮点）
PRV(881) #2 #0 D804  ; 右机械手当前位置脉冲
FLTL(453) D804 D806  ; 右机械手当前位置脉冲, 右机械手当前位置脉冲(浮点)
/F(457) D806 D802 D808  ; 右机械手当前位置脉冲(浮点), 右机械手脉冲当量(浮点）, 右机械手当前位置(mm)

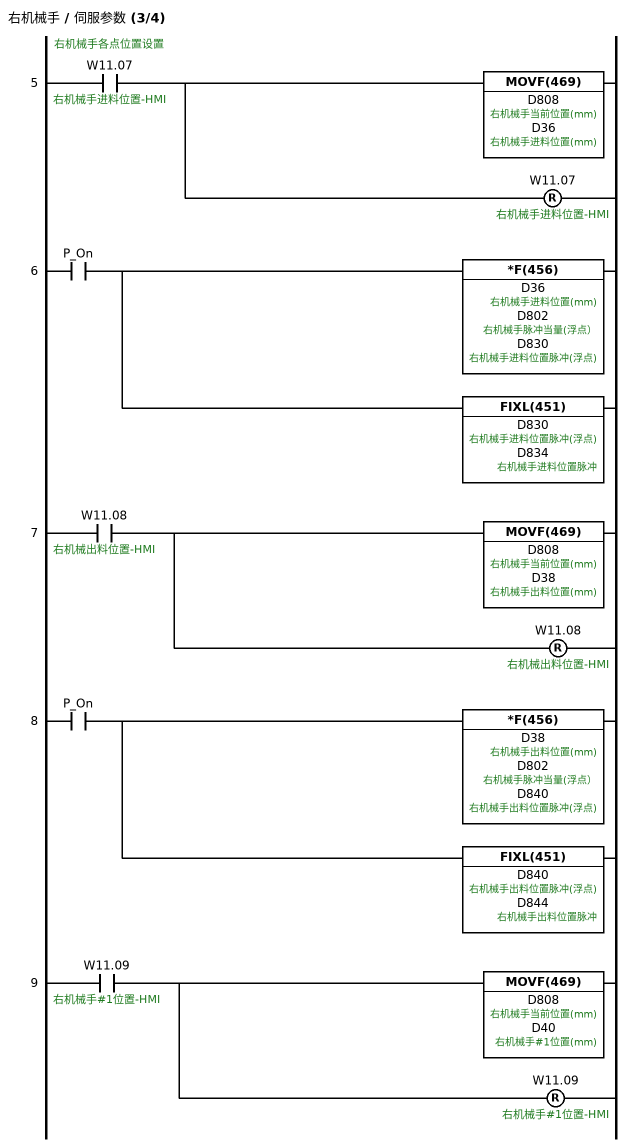
; rung 5: 右机械手各点位置设置
LD W11.07  ; 右机械手进料位置-HMI
MOVF(469) D808 D36  ; 右机械手当前位置(mm), 右机械手进料位置(mm)
RSET W11.07  ; 右机械手进料位置-HMI
; rung 6
LD P_On
*F(456) D36 D802 D830  ; 右机械手进料位置(mm), 右机械手脉冲当量(浮点）, 右机械手进料位置脉冲(浮点)
FIXL(451) D830 D834  ; 右机械手进料位置脉冲(浮点), 右机械手进料位置脉冲
; rung 7
LD W11.08  ; 右机械出料位置-HMI
MOVF(469) D808 D38  ; 右机械手当前位置(mm), 右机械手出料位置(mm)
RSET W11.08  ; 右机械出料位置-HMI
; rung 8
LD P_On
*F(456) D38 D802 D840  ; 右机械手出料位置(mm), 右机械手脉冲当量(浮点）, 右机械手出料位置脉冲(浮点)
FIXL(451) D840 D844  ; 右机械手出料位置脉冲(浮点), 右机械手出料位置脉冲
; rung 9
LD W11.09  ; 右机械手#1位置-HMI
MOVF(469) D808 D40  ; 右机械手当前位置(mm), 右机械手#1位置(mm)
RSET W11.09  ; 右机械手#1位置-HMI

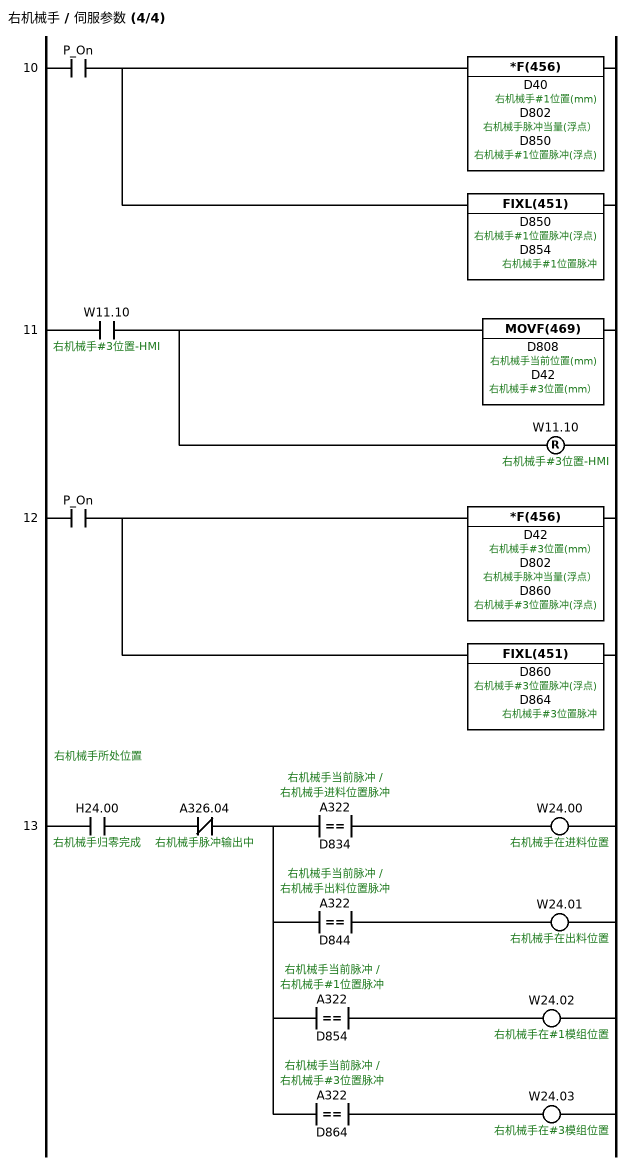
; rung 10
LD P_On
*F(456) D40 D802 D850  ; 右机械手#1位置(mm), 右机械手脉冲当量(浮点）, 右机械手#1位置脉冲(浮点)
FIXL(451) D850 D854  ; 右机械手#1位置脉冲(浮点), 右机械手#1位置脉冲
; rung 11
LD W11.10  ; 右机械手#3位置-HMI
MOVF(469) D808 D42  ; 右机械手当前位置(mm), 右机械手#3位置(mm）
RSET W11.10  ; 右机械手#3位置-HMI
; rung 12
LD P_On
*F(456) D42 D802 D860  ; 右机械手#3位置(mm）, 右机械手脉冲当量(浮点）, 右机械手#3位置脉冲(浮点)
FIXL(451) D860 D864  ; 右机械手#3位置脉冲(浮点), 右机械手#3位置脉冲
; rung 13: 右机械手所处位置
LD H24.00  ; 右机械手归零完成
ANDNOT A326.04  ; 右机械手脉冲输出中
OUT TR0
AND=SL(303) A322 D834  ; 右机械手当前脉冲, 右机械手进料位置脉冲
OUT W24.00  ; 右机械手在进料位置
LD TR0
AND=SL(303) A322 D844  ; 右机械手当前脉冲, 右机械手出料位置脉冲
OUT W24.01  ; 右机械手在出料位置
LD TR0
AND=SL(303) A322 D854  ; 右机械手当前脉冲, 右机械手#1位置脉冲
OUT W24.02  ; 右机械手在#1模组位置
LD TR0
AND=SL(303) A322 D864  ; 右机械手当前脉冲, 右机械手#3位置脉冲
OUT W24.03  ; 右机械手在#3模组位置

### Section 轴控运动及外部输出

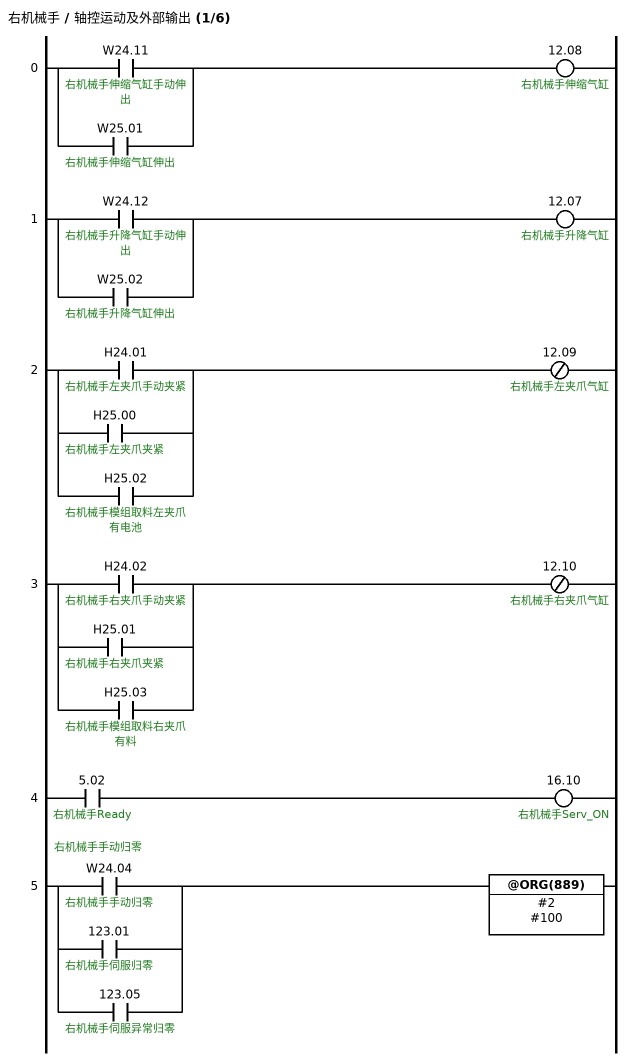
; rung 0
LD W24.11  ; 右机械手伸缩气缸手动伸出
OR W25.01  ; 右机械手伸缩气缸伸出
OUT 12.08  ; 右机械手伸缩气缸
; rung 1
LD W24.12  ; 右机械手升降气缸手动伸出
OR W25.02  ; 右机械手升降气缸伸出
OUT 12.07  ; 右机械手升降气缸
; rung 2
LD H24.01  ; 右机械手左夹爪手动夹紧
OR H25.00  ; 右机械手左夹爪夹紧
OR H25.02  ; 右机械手模组取料左夹爪有电池
OUTNOT 12.09  ; 右机械手左夹爪气缸
; rung 3
LD H24.02  ; 右机械手右夹爪手动夹紧
OR H25.01  ; 右机械手右夹爪夹紧
OR H25.03  ; 右机械手模组取料右夹爪有料
OUTNOT 12.10  ; 右机械手右夹爪气缸
; rung 4
LD 5.02  ; 右机械手Ready
OUT 16.10  ; 右机械手Serv_ON
; rung 5: 右机械手手动归零
LD W24.04  ; 右机械手手动归零
OR 123.01  ; 右机械手伺服归零
OR 123.05  ; 右机械手伺服异常归零
@ORG(889) #2 #100

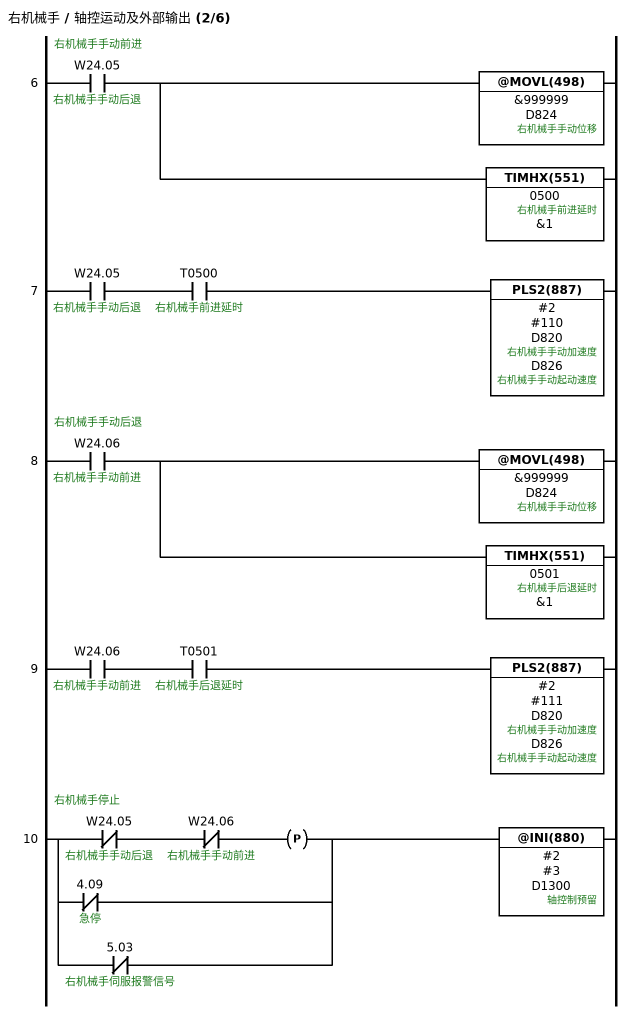
; rung 6: 右机械手手动前进
LD W24.05  ; 右机械手手动后退
@MOVL(498) &999999 D824  ; 右机械手手动位移
TIMHX(551) 0500 &1  ; 右机械手前进延时
; rung 7
LD W24.05  ; 右机械手手动后退
AND T0500  ; 右机械手前进延时
PLS2(887) #2 #110 D820 D826  ; 右机械手手动加速度, 右机械手手动起动速度
; rung 8: 右机械手手动后退
LD W24.06  ; 右机械手手动前进
@MOVL(498) &999999 D824  ; 右机械手手动位移
TIMHX(551) 0501 &1  ; 右机械手后退延时
; rung 9
LD W24.06  ; 右机械手手动前进
AND T0501  ; 右机械手后退延时
PLS2(887) #2 #111 D820 D826  ; 右机械手手动加速度, 右机械手手动起动速度
; rung 10: 右机械手停止
LDNOT W24.05  ; 右机械手手动后退
ANDNOT W24.06  ; 右机械手手动前进
UP(521)
ORNOT 4.09  ; 急停
ORNOT 5.03  ; 右机械手伺服报警信号
@INI(880) #2 #3 D1300  ; 轴控制预留

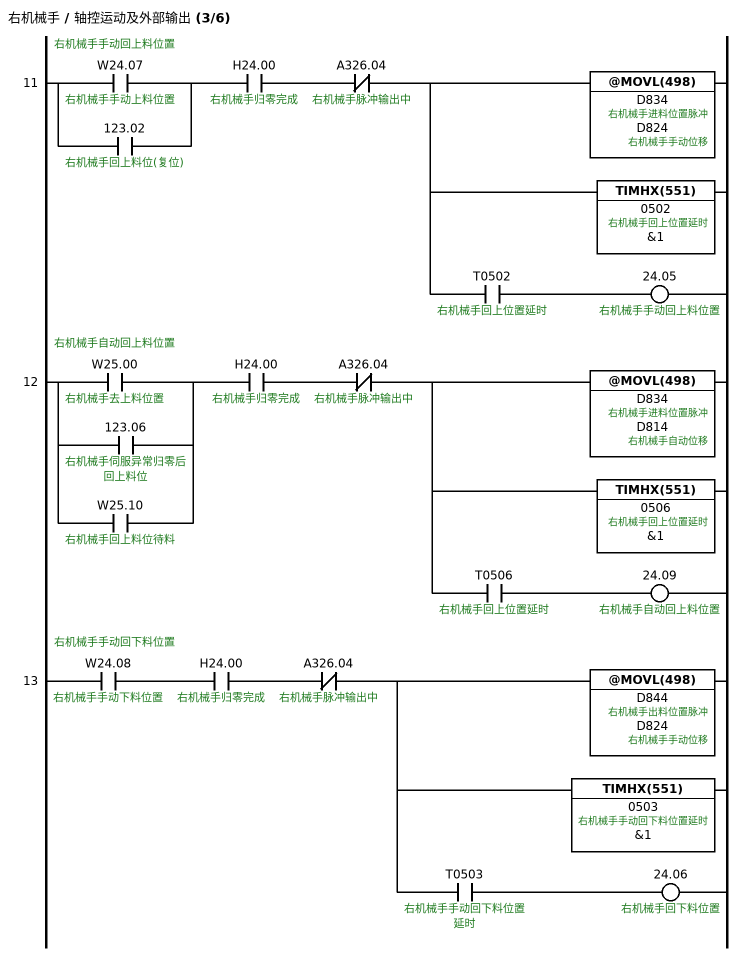
; rung 11: 右机械手手动回上料位置
LD W24.07  ; 右机械手手动上料位置
OR 123.02  ; 右机械手回上料位(复位)
AND H24.00  ; 右机械手归零完成
ANDNOT A326.04  ; 右机械手脉冲输出中
@MOVL(498) D834 D824  ; 右机械手进料位置脉冲, 右机械手手动位移
TIMHX(551) 0502 &1  ; 右机械手回上位置延时
AND T0502  ; 右机械手回上位置延时
OUT 24.05  ; 右机械手手动回上料位置
; rung 12: 右机械手自动回上料位置
LD W25.00  ; 右机械手去上料位置
OR 123.06  ; 右机械手伺服异常归零后回上料位
OR W25.10  ; 右机械手回上料位待料
AND H24.00  ; 右机械手归零完成
ANDNOT A326.04  ; 右机械手脉冲输出中
@MOVL(498) D834 D814  ; 右机械手进料位置脉冲, 右机械手自动位移
TIMHX(551) 0506 &1  ; 右机械手回上位置延时
AND T0506  ; 右机械手回上位置延时
OUT 24.09  ; 右机械手自动回上料位置
; rung 13: 右机械手手动回下料位置
LD W24.08  ; 右机械手手动下料位置
AND H24.00  ; 右机械手归零完成
ANDNOT A326.04  ; 右机械手脉冲输出中
@MOVL(498) D844 D824  ; 右机械手出料位置脉冲, 右机械手手动位移
TIMHX(551) 0503 &1  ; 右机械手手动回下料位置延时
AND T0503  ; 右机械手手动回下料位置延时
OUT 24.06  ; 右机械手回下料位置

